FUNCTION_BLOCK FB_System_HOWW_261
VAR_INPUT
	Freigabe_auto			: BOOL;
	Freigabe_Deakt_auto		: BOOL;
	Betrieb_Anford_auto		: BOOL;
	HO_Zustand				: ST_HO_Zustand;
	HO_Parameter			: ST_HO_Parameter;
END_VAR
VAR_OUTPUT
	{attribute 'OPC.UA.DA' := '1'}Steuerung				: ST_System_HOWW_Steuerung;			
	{attribute 'OPC.UA.DA' := '1'}Stellwert				: ST_System_HOWW_Stellwert;			
	{attribute 'OPC.UA.DA' := '1'}Zustand					: ST_System_HOWW_Zustand;		
	{attribute 'OPC.UA.DA' := '1'}Parameter				: ST_System_HOWW_Parameter;			
END_VAR
VAR
	Pumpe_261				: FB_PU;
	Stellventil_261			: FB_SVs;
	Regelventil_261			: FB_RV; (*neu 14.07.2020*)

	Zustandscheck			: FB_System_HOWW_Zustandscheck;
	Logik					: FB_System_HOWW_Logik;
	Ablaufsteuerung			: FB_System_HOWW_Ablaufsteuerung;
END_VAR
VAR // added by the converter: edge detectors and wires of the graphical bodies
    _w1 : ANY;
END_VAR

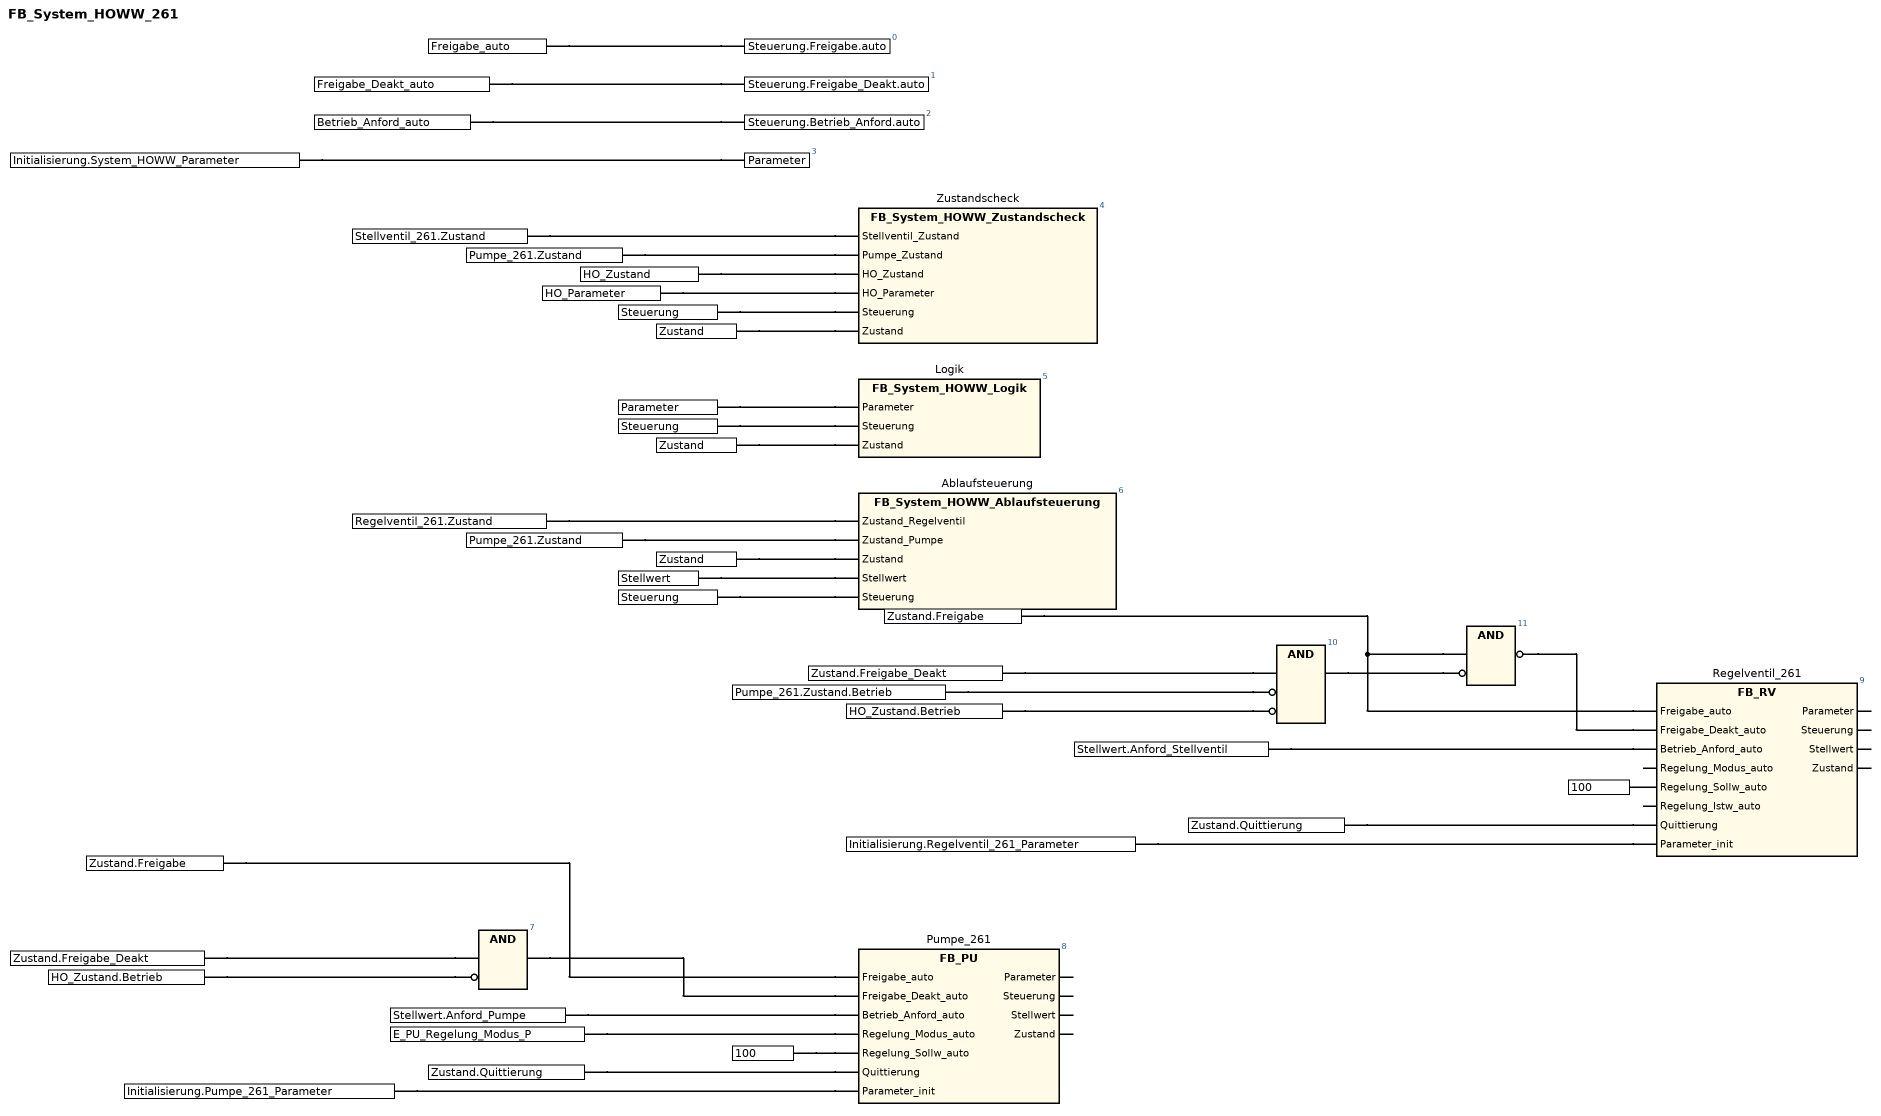
Steuerung.Freigabe.auto := Freigabe_auto;
Steuerung.Freigabe_Deakt.auto := Freigabe_Deakt_auto;
Steuerung.Betrieb_Anford.auto := Betrieb_Anford_auto;
Parameter := Initialisierung.System_HOWW_Parameter;
Zustandscheck(
    Stellventil_Zustand := Stellventil_261.Zustand,
    Pumpe_Zustand := Pumpe_261.Zustand,
    HO_Zustand := HO_Zustand,
    HO_Parameter := HO_Parameter,
    Steuerung := Steuerung,
    Zustand := Zustand); // FB_System_HOWW_Zustandscheck
Logik(Parameter := Parameter, Steuerung := Steuerung, Zustand := Zustand); // FB_System_HOWW_Logik
Ablaufsteuerung(
    Zustand_Regelventil := Regelventil_261.Zustand,
    Zustand_Pumpe := Pumpe_261.Zustand,
    Zustand := Zustand,
    Stellwert := Stellwert,
    Steuerung := Steuerung); // FB_System_HOWW_Ablaufsteuerung
Pumpe_261(
    Freigabe_auto := Zustand.Freigabe,
    Freigabe_Deakt_auto := Zustand.Freigabe_Deakt AND NOT HO_Zustand.Betrieb,
    Betrieb_Anford_auto := Stellwert.Anford_Pumpe,
    Regelung_Modus_auto := E_PU_Regelung_Modus_P,
    Regelung_Sollw_auto := 100,
    Quittierung := Zustand.Quittierung,
    Parameter_init := Initialisierung.Pumpe_261_Parameter); // FB_PU
Regelventil_261(
    Freigabe_auto := Zustand.Freigabe,
    Freigabe_Deakt_auto := NOT _w1,
    Betrieb_Anford_auto := Stellwert.Anford_Stellventil,
    Regelung_Sollw_auto := 100,
    Quittierung := Zustand.Quittierung,
    Parameter_init := Initialisierung.Regelventil_261_Parameter); // FB_RV
_w1 := Zustand.Freigabe AND NOT (Zustand.Freigabe_Deakt AND NOT Pumpe_261.Zustand.Betrieb AND NOT HO_Zustand.Betrieb);

END_FUNCTION_BLOCK

(* stored: Version 1.1.0.1, ProductVersion 3.1.4024.9
   POU FB_System_HOWW_261: Id {632ed535-050c-4b43-8772-bec79f160240}, SpecialFunc None *)
